TYPE
	jog_manager_test_command_enum: (
	JOG_MANAGER_TEST_CMD_NONE				:= 0	(*$ No command assigned $*)
	) := JOG_MANAGER_TEST_CMD_NONE;
END_TYPE

(* stored: Version 1.1.0.1, ProductVersion 3.1.4022.12
   DUT jog_manager_test_command_enum: Id {6f201085-9960-4461-85f4-bcfa1654387d} *)
